(* Logix 5000 project; controller cal1632 1756-L62 rev 16.20; software revision 16.05; part 47 of 57 *)
(* tags used below, declared in another part *)
   FAULT : BOOL;
   HMI : BOOL;
   p01r09_pb_global_reset : BOOL;
   p02_dint_from_hmi : hmi_dint;
   p27_ao_dia_a : REAL;
   p27_ao_dia_b : REAL;
   p27_dint_to_hmi : DINT[16];
   p27_real_to_hmi : REAL[112];
   p27r05_lla_mode_tension : BOOL;
   p27r05_llb_mode_tension : BOOL;
   p27r06 : routine;
   p27r06_timer_fault : TIMER[4];
   p27r06_timer_warning : TIMER[4];
   p27r07 : routine;
   p27r07_timer_fault : TIMER[4];
   p27r07_timer_warning : TIMER[4];
   p27r08 : routine;
   p27r08_timer_fault : TIMER[4];
   p27r08_timer_warning : TIMER[4];
   p27r09 : routine;
   p27r09_a_enable_toggle : SYS_Toggle;
   p27r09_b_enable_toggle : SYS_Toggle;
   p27r09_timer_fault : TIMER[4];
   p27r09_timer_warning : TIMER[4];
(* P27_Lower_Poly_Letoff, continued *)

ROUTINE R06_Real_to_HMI   (* ladder *)
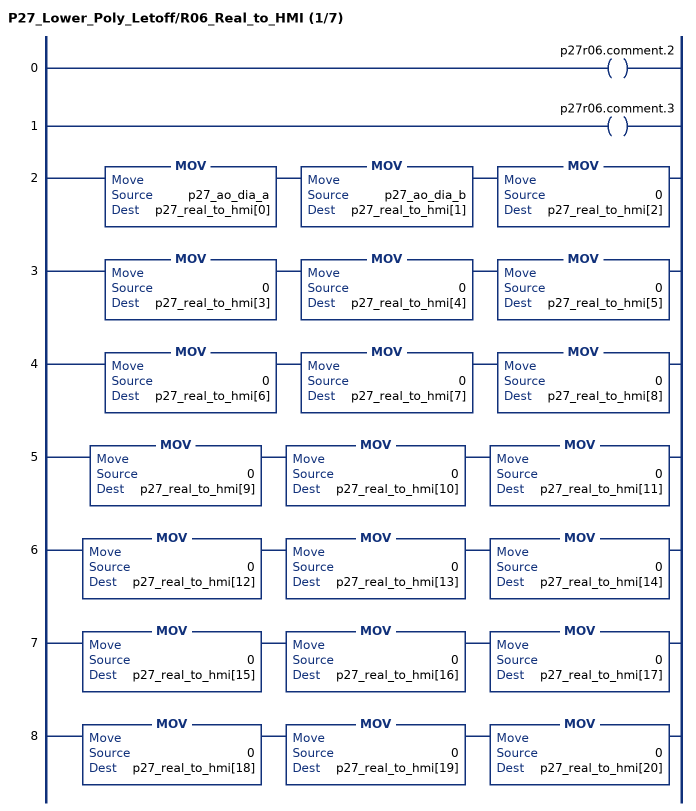
   0: OTE(p27r06.comment.2);
   1: OTE(p27r06.comment.3);
   2: MOV(p27_ao_dia_a,p27_real_to_hmi[0])MOV(p27_ao_dia_b,p27_real_to_hmi[1])MOV(0,p27_real_to_hmi[2]);
   3: MOV(0,p27_real_to_hmi[3])MOV(0,p27_real_to_hmi[4])MOV(0,p27_real_to_hmi[5]);
   4: MOV(0,p27_real_to_hmi[6])MOV(0,p27_real_to_hmi[7])MOV(0,p27_real_to_hmi[8]);
   5: MOV(0,p27_real_to_hmi[9])MOV(0,p27_real_to_hmi[10])MOV(0,p27_real_to_hmi[11]);
   6: MOV(0,p27_real_to_hmi[12])MOV(0,p27_real_to_hmi[13])MOV(0,p27_real_to_hmi[14]);
   7: MOV(0,p27_real_to_hmi[15])MOV(0,p27_real_to_hmi[16])MOV(0,p27_real_to_hmi[17]);
   8: MOV(0,p27_real_to_hmi[18])MOV(0,p27_real_to_hmi[19])MOV(0,p27_real_to_hmi[20]);
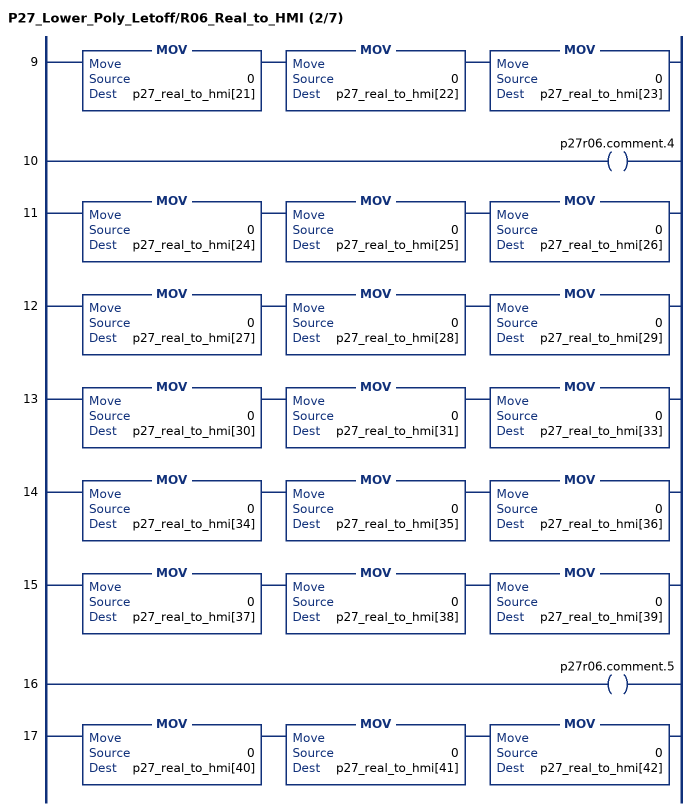
   9: MOV(0,p27_real_to_hmi[21])MOV(0,p27_real_to_hmi[22])MOV(0,p27_real_to_hmi[23]);
   10: OTE(p27r06.comment.4);
   11: MOV(0,p27_real_to_hmi[24])MOV(0,p27_real_to_hmi[25])MOV(0,p27_real_to_hmi[26]);
   12: MOV(0,p27_real_to_hmi[27])MOV(0,p27_real_to_hmi[28])MOV(0,p27_real_to_hmi[29]);
   13: MOV(0,p27_real_to_hmi[30])MOV(0,p27_real_to_hmi[31])MOV(0,p27_real_to_hmi[33]);
   14: MOV(0,p27_real_to_hmi[34])MOV(0,p27_real_to_hmi[35])MOV(0,p27_real_to_hmi[36]);
   15: MOV(0,p27_real_to_hmi[37])MOV(0,p27_real_to_hmi[38])MOV(0,p27_real_to_hmi[39]);
   16: OTE(p27r06.comment.5);
   17: MOV(0,p27_real_to_hmi[40])MOV(0,p27_real_to_hmi[41])MOV(0,p27_real_to_hmi[42]);
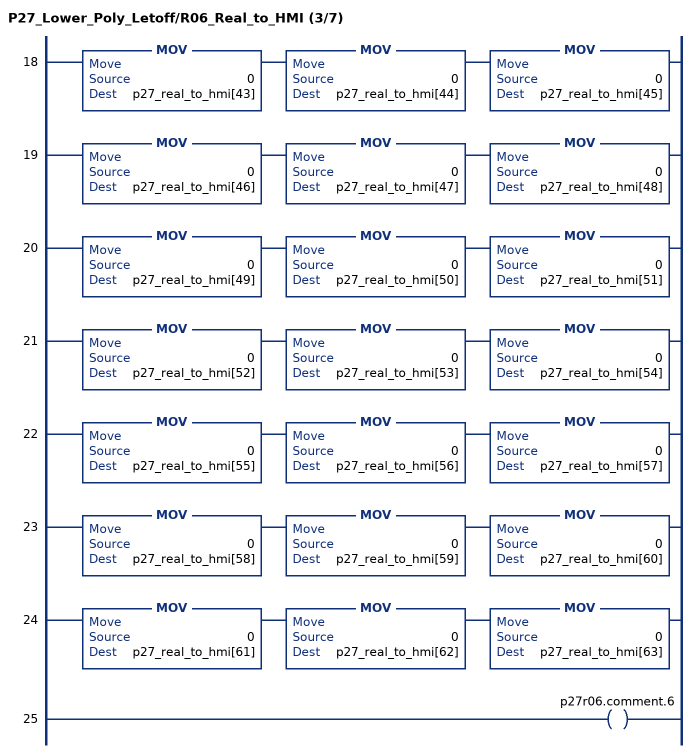
   18: MOV(0,p27_real_to_hmi[43])MOV(0,p27_real_to_hmi[44])MOV(0,p27_real_to_hmi[45]);
   19: MOV(0,p27_real_to_hmi[46])MOV(0,p27_real_to_hmi[47])MOV(0,p27_real_to_hmi[48]);
   20: MOV(0,p27_real_to_hmi[49])MOV(0,p27_real_to_hmi[50])MOV(0,p27_real_to_hmi[51]);
   21: MOV(0,p27_real_to_hmi[52])MOV(0,p27_real_to_hmi[53])MOV(0,p27_real_to_hmi[54]);
   22: MOV(0,p27_real_to_hmi[55])MOV(0,p27_real_to_hmi[56])MOV(0,p27_real_to_hmi[57]);
   23: MOV(0,p27_real_to_hmi[58])MOV(0,p27_real_to_hmi[59])MOV(0,p27_real_to_hmi[60]);
   24: MOV(0,p27_real_to_hmi[61])MOV(0,p27_real_to_hmi[62])MOV(0,p27_real_to_hmi[63]);
   25: OTE(p27r06.comment.6);
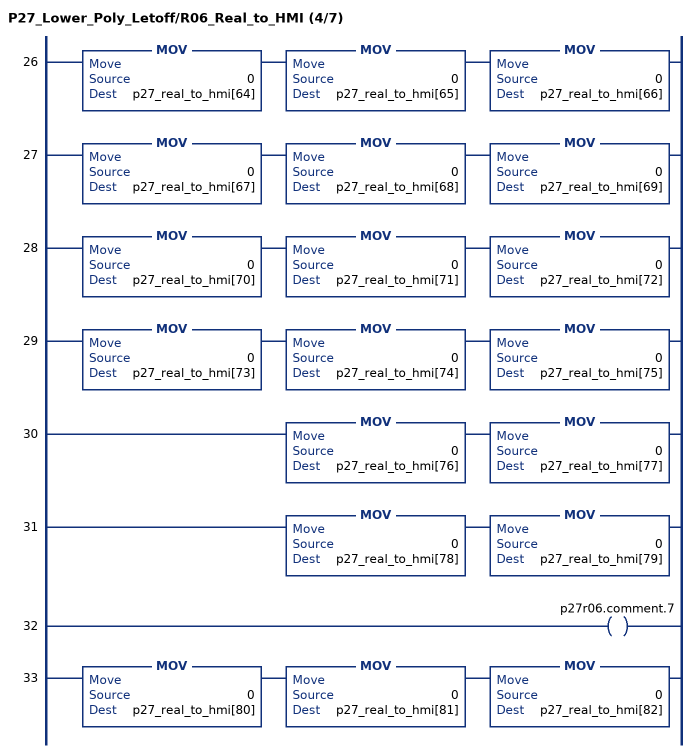
   26: MOV(0,p27_real_to_hmi[64])MOV(0,p27_real_to_hmi[65])MOV(0,p27_real_to_hmi[66]);
   27: MOV(0,p27_real_to_hmi[67])MOV(0,p27_real_to_hmi[68])MOV(0,p27_real_to_hmi[69]);
   28: MOV(0,p27_real_to_hmi[70])MOV(0,p27_real_to_hmi[71])MOV(0,p27_real_to_hmi[72]);
   29: MOV(0,p27_real_to_hmi[73])MOV(0,p27_real_to_hmi[74])MOV(0,p27_real_to_hmi[75]);
   30: MOV(0,p27_real_to_hmi[76])MOV(0,p27_real_to_hmi[77]);
   31: MOV(0,p27_real_to_hmi[78])MOV(0,p27_real_to_hmi[79]);
   32: OTE(p27r06.comment.7);
   33: MOV(0,p27_real_to_hmi[80])MOV(0,p27_real_to_hmi[81])MOV(0,p27_real_to_hmi[82]);
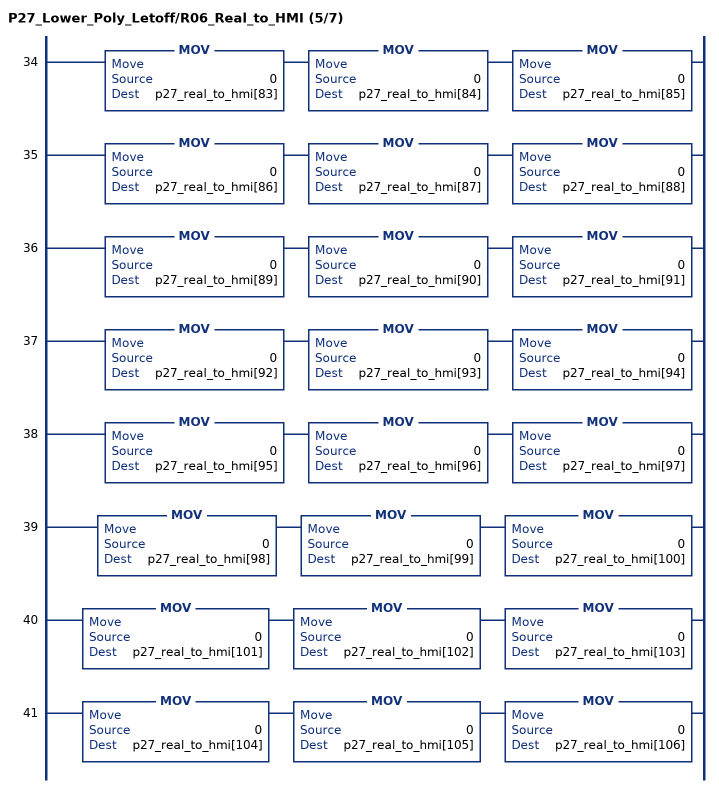
   34: MOV(0,p27_real_to_hmi[83])MOV(0,p27_real_to_hmi[84])MOV(0,p27_real_to_hmi[85]);
   35: MOV(0,p27_real_to_hmi[86])MOV(0,p27_real_to_hmi[87])MOV(0,p27_real_to_hmi[88]);
   36: MOV(0,p27_real_to_hmi[89])MOV(0,p27_real_to_hmi[90])MOV(0,p27_real_to_hmi[91]);
   37: MOV(0,p27_real_to_hmi[92])MOV(0,p27_real_to_hmi[93])MOV(0,p27_real_to_hmi[94]);
   38: MOV(0,p27_real_to_hmi[95])MOV(0,p27_real_to_hmi[96])MOV(0,p27_real_to_hmi[97]);
   39: MOV(0,p27_real_to_hmi[98])MOV(0,p27_real_to_hmi[99])MOV(0,p27_real_to_hmi[100]);
   40: MOV(0,p27_real_to_hmi[101])MOV(0,p27_real_to_hmi[102])MOV(0,p27_real_to_hmi[103]);
   41: MOV(0,p27_real_to_hmi[104])MOV(0,p27_real_to_hmi[105])MOV(0,p27_real_to_hmi[106]);
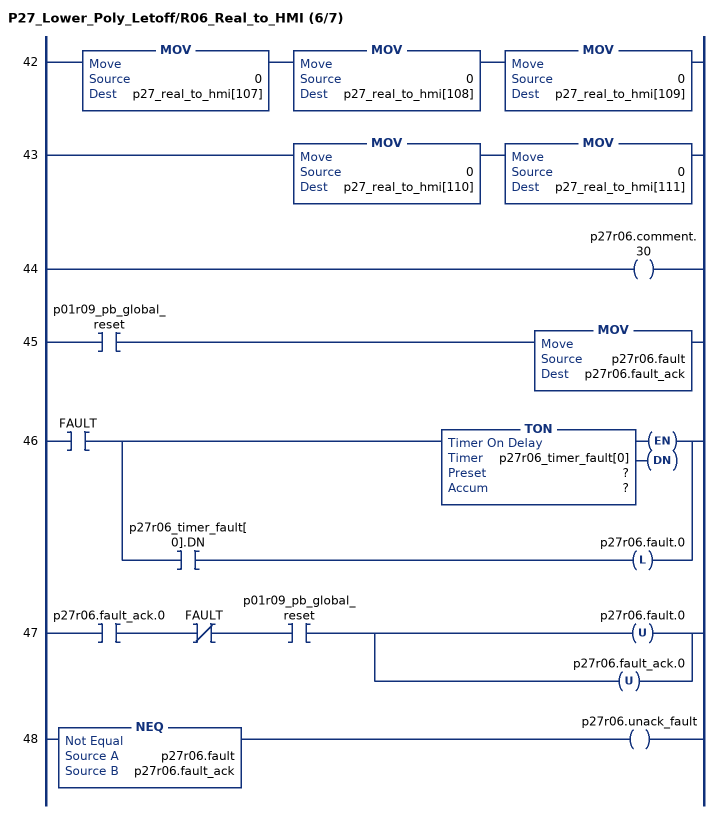
   42: MOV(0,p27_real_to_hmi[107])MOV(0,p27_real_to_hmi[108])MOV(0,p27_real_to_hmi[109]);
   43: MOV(0,p27_real_to_hmi[110])MOV(0,p27_real_to_hmi[111]);
   44: OTE(p27r06.comment.30);
   45: XIC(p01r09_pb_global_reset)MOV(p27r06.fault,p27r06.fault_ack);
   46: XIC(FAULT)[TON(p27r06_timer_fault[0],?,?) ,XIC(p27r06_timer_fault[0].DN) OTL(p27r06.fault.0) ];
   47: XIC(p27r06.fault_ack.0)XIO(FAULT)XIC(p01r09_pb_global_reset)[OTU(p27r06.fault.0) ,OTU(p27r06.fault_ack.0) ];
   48: NEQ(p27r06.fault,p27r06.fault_ack)OTE(p27r06.unack_fault);
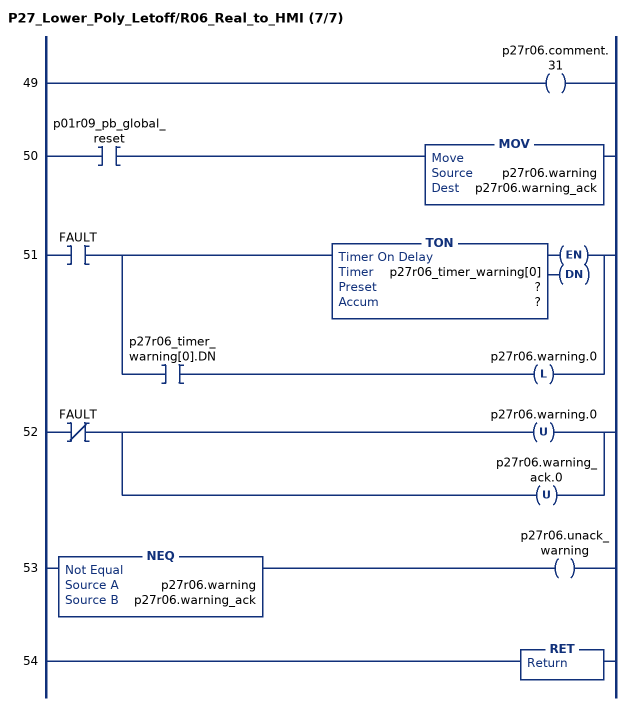
   49: OTE(p27r06.comment.31);
   50: XIC(p01r09_pb_global_reset)MOV(p27r06.warning,p27r06.warning_ack);
   51: XIC(FAULT)[TON(p27r06_timer_warning[0],?,?) ,XIC(p27r06_timer_warning[0].DN) OTL(p27r06.warning.0) ];
   52: XIO(FAULT)[OTU(p27r06.warning.0) ,OTU(p27r06.warning_ack.0) ];
   53: NEQ(p27r06.warning,p27r06.warning_ack)OTE(p27r06.unack_warning);
   54: RET();
END_ROUTINE

ROUTINE R07_Alarms   (* ladder *)
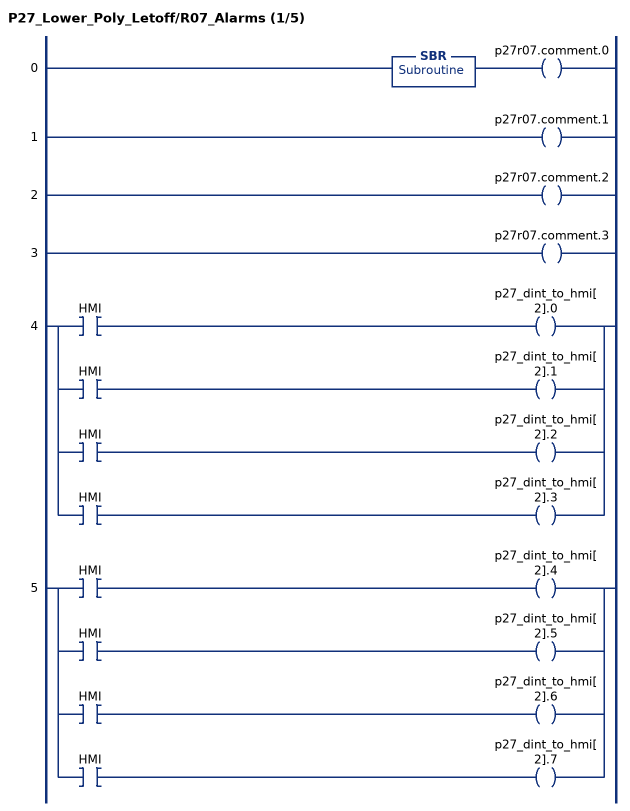
   0: SBR()OTE(p27r07.comment.0);
   1: OTE(p27r07.comment.1);
   2: OTE(p27r07.comment.2);
   3: OTE(p27r07.comment.3);
   4: [XIC(HMI) OTE(p27_dint_to_hmi[2].0) ,XIC(HMI) OTE(p27_dint_to_hmi[2].1) ,XIC(HMI) OTE(p27_dint_to_hmi[2].2) ,XIC(HMI) OTE(p27_dint_to_hmi[2].3) ];
   5: [XIC(HMI) OTE(p27_dint_to_hmi[2].4) ,XIC(HMI) OTE(p27_dint_to_hmi[2].5) ,XIC(HMI) OTE(p27_dint_to_hmi[2].6) ,XIC(HMI) OTE(p27_dint_to_hmi[2].7) ];
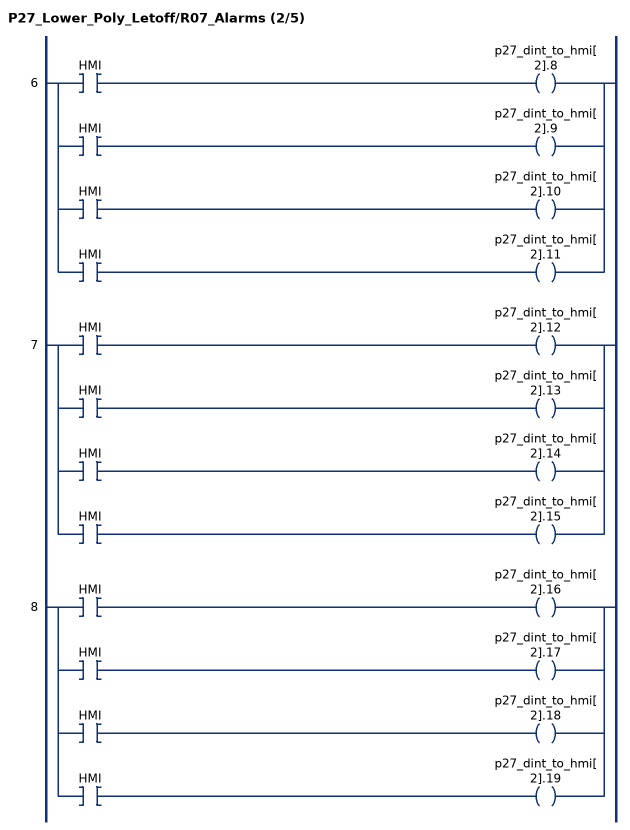
   6: [XIC(HMI) OTE(p27_dint_to_hmi[2].8) ,XIC(HMI) OTE(p27_dint_to_hmi[2].9) ,XIC(HMI) OTE(p27_dint_to_hmi[2].10) ,XIC(HMI) OTE(p27_dint_to_hmi[2].11) ];
   7: [XIC(HMI) OTE(p27_dint_to_hmi[2].12) ,XIC(HMI) OTE(p27_dint_to_hmi[2].13) ,XIC(HMI) OTE(p27_dint_to_hmi[2].14) ,XIC(HMI) OTE(p27_dint_to_hmi[2].15) ];
   8: [XIC(HMI) OTE(p27_dint_to_hmi[2].16) ,XIC(HMI) OTE(p27_dint_to_hmi[2].17) ,XIC(HMI) OTE(p27_dint_to_hmi[2].18) ,XIC(HMI) OTE(p27_dint_to_hmi[2].19) ];
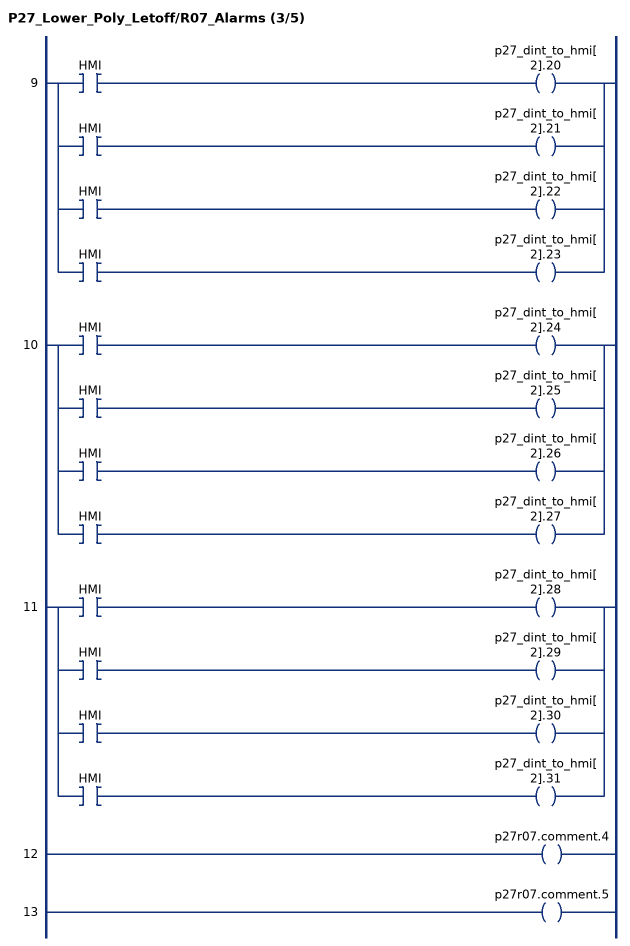
   9: [XIC(HMI) OTE(p27_dint_to_hmi[2].20) ,XIC(HMI) OTE(p27_dint_to_hmi[2].21) ,XIC(HMI) OTE(p27_dint_to_hmi[2].22) ,XIC(HMI) OTE(p27_dint_to_hmi[2].23) ];
   10: [XIC(HMI) OTE(p27_dint_to_hmi[2].24) ,XIC(HMI) OTE(p27_dint_to_hmi[2].25) ,XIC(HMI) OTE(p27_dint_to_hmi[2].26) ,XIC(HMI) OTE(p27_dint_to_hmi[2].27) ];
   11: [XIC(HMI) OTE(p27_dint_to_hmi[2].28) ,XIC(HMI) OTE(p27_dint_to_hmi[2].29) ,XIC(HMI) OTE(p27_dint_to_hmi[2].30) ,XIC(HMI) OTE(p27_dint_to_hmi[2].31) ];
   12: OTE(p27r07.comment.4);
   13: OTE(p27r07.comment.5);
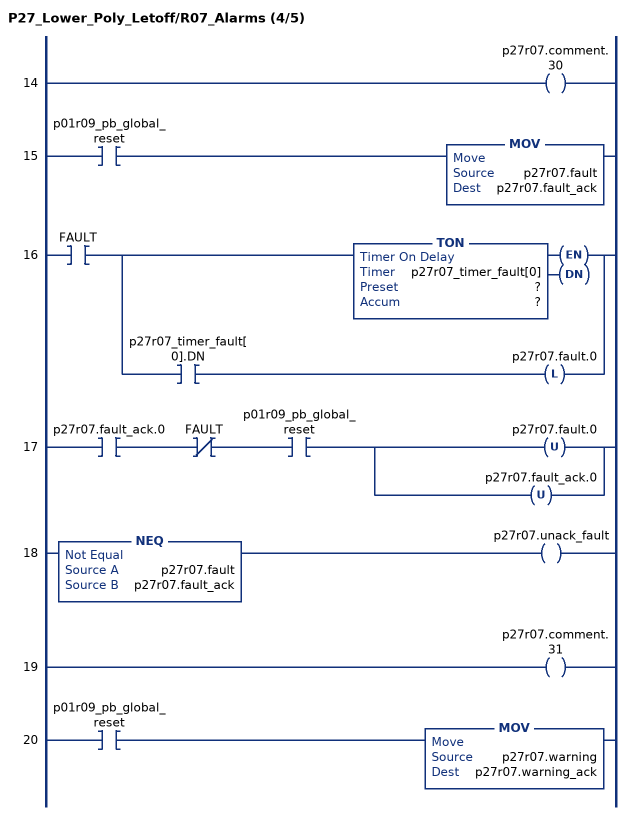
   14: OTE(p27r07.comment.30);
   15: XIC(p01r09_pb_global_reset)MOV(p27r07.fault,p27r07.fault_ack);
   16: XIC(FAULT)[TON(p27r07_timer_fault[0],?,?) ,XIC(p27r07_timer_fault[0].DN) OTL(p27r07.fault.0) ];
   17: XIC(p27r07.fault_ack.0)XIO(FAULT)XIC(p01r09_pb_global_reset)[OTU(p27r07.fault.0) ,OTU(p27r07.fault_ack.0) ];
   18: NEQ(p27r07.fault,p27r07.fault_ack)OTE(p27r07.unack_fault);
   19: OTE(p27r07.comment.31);
   20: XIC(p01r09_pb_global_reset)MOV(p27r07.warning,p27r07.warning_ack);
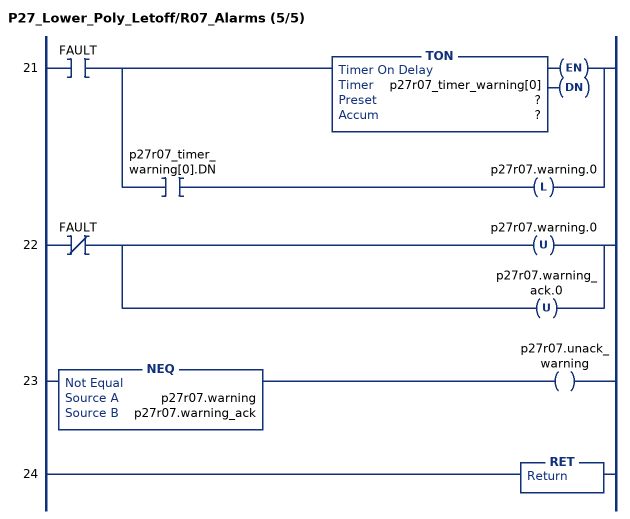
   21: XIC(FAULT)[TON(p27r07_timer_warning[0],?,?) ,XIC(p27r07_timer_warning[0].DN) OTL(p27r07.warning.0) ];
   22: XIO(FAULT)[OTU(p27r07.warning.0) ,OTU(p27r07.warning_ack.0) ];
   23: NEQ(p27r07.warning,p27r07.warning_ack)OTE(p27r07.unack_warning);
   24: RET();
END_ROUTINE

ROUTINE R08_Warnings   (* ladder *)
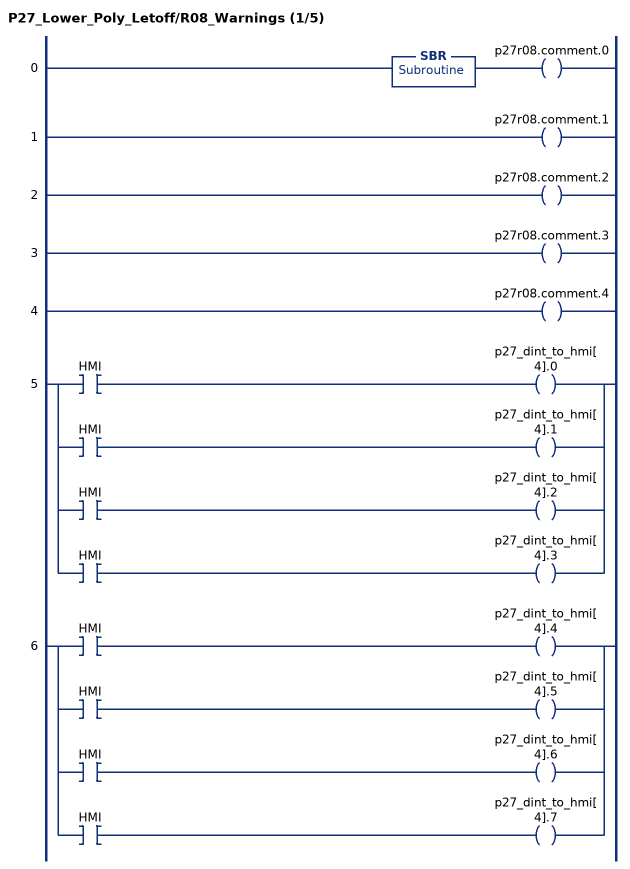
   0: SBR()OTE(p27r08.comment.0);
   1: OTE(p27r08.comment.1);
   2: OTE(p27r08.comment.2);
   3: OTE(p27r08.comment.3);
   4: OTE(p27r08.comment.4);
   5: [XIC(HMI) OTE(p27_dint_to_hmi[4].0) ,XIC(HMI) OTE(p27_dint_to_hmi[4].1) ,XIC(HMI) OTE(p27_dint_to_hmi[4].2) ,XIC(HMI) OTE(p27_dint_to_hmi[4].3) ];
   6: [XIC(HMI) OTE(p27_dint_to_hmi[4].4) ,XIC(HMI) OTE(p27_dint_to_hmi[4].5) ,XIC(HMI) OTE(p27_dint_to_hmi[4].6) ,XIC(HMI) OTE(p27_dint_to_hmi[4].7) ];
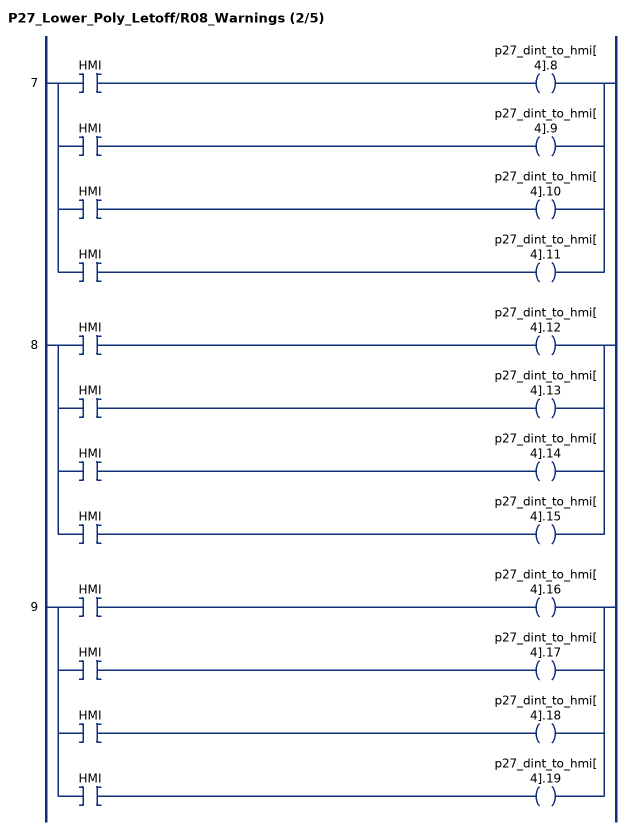
   7: [XIC(HMI) OTE(p27_dint_to_hmi[4].8) ,XIC(HMI) OTE(p27_dint_to_hmi[4].9) ,XIC(HMI) OTE(p27_dint_to_hmi[4].10) ,XIC(HMI) OTE(p27_dint_to_hmi[4].11) ];
   8: [XIC(HMI) OTE(p27_dint_to_hmi[4].12) ,XIC(HMI) OTE(p27_dint_to_hmi[4].13) ,XIC(HMI) OTE(p27_dint_to_hmi[4].14) ,XIC(HMI) OTE(p27_dint_to_hmi[4].15) ];
   9: [XIC(HMI) OTE(p27_dint_to_hmi[4].16) ,XIC(HMI) OTE(p27_dint_to_hmi[4].17) ,XIC(HMI) OTE(p27_dint_to_hmi[4].18) ,XIC(HMI) OTE(p27_dint_to_hmi[4].19) ];
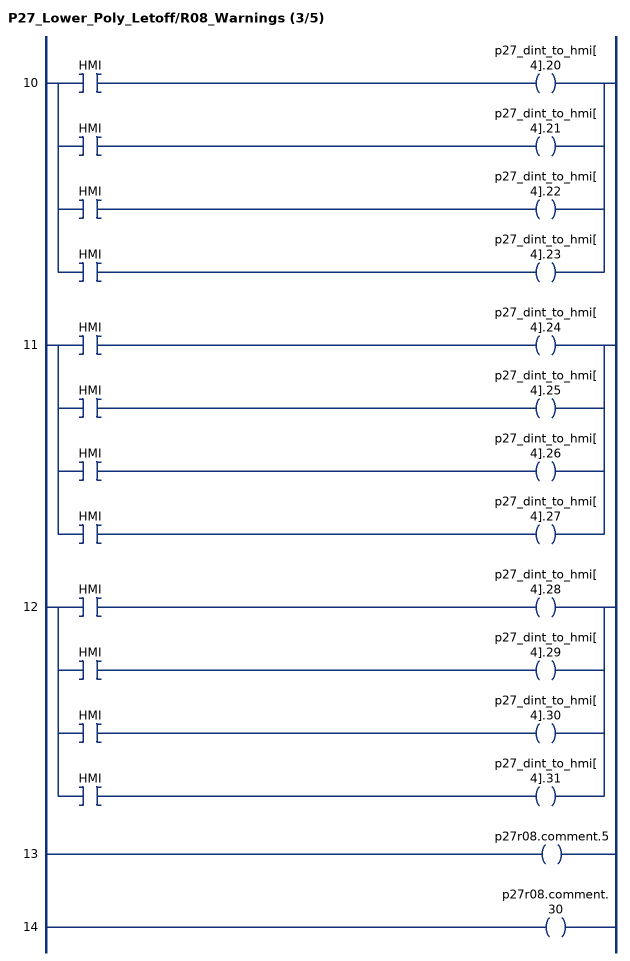
   10: [XIC(HMI) OTE(p27_dint_to_hmi[4].20) ,XIC(HMI) OTE(p27_dint_to_hmi[4].21) ,XIC(HMI) OTE(p27_dint_to_hmi[4].22) ,XIC(HMI) OTE(p27_dint_to_hmi[4].23) ];
   11: [XIC(HMI) OTE(p27_dint_to_hmi[4].24) ,XIC(HMI) OTE(p27_dint_to_hmi[4].25) ,XIC(HMI) OTE(p27_dint_to_hmi[4].26) ,XIC(HMI) OTE(p27_dint_to_hmi[4].27) ];
   12: [XIC(HMI) OTE(p27_dint_to_hmi[4].28) ,XIC(HMI) OTE(p27_dint_to_hmi[4].29) ,XIC(HMI) OTE(p27_dint_to_hmi[4].30) ,XIC(HMI) OTE(p27_dint_to_hmi[4].31) ];
   13: OTE(p27r08.comment.5);
   14: OTE(p27r08.comment.30);
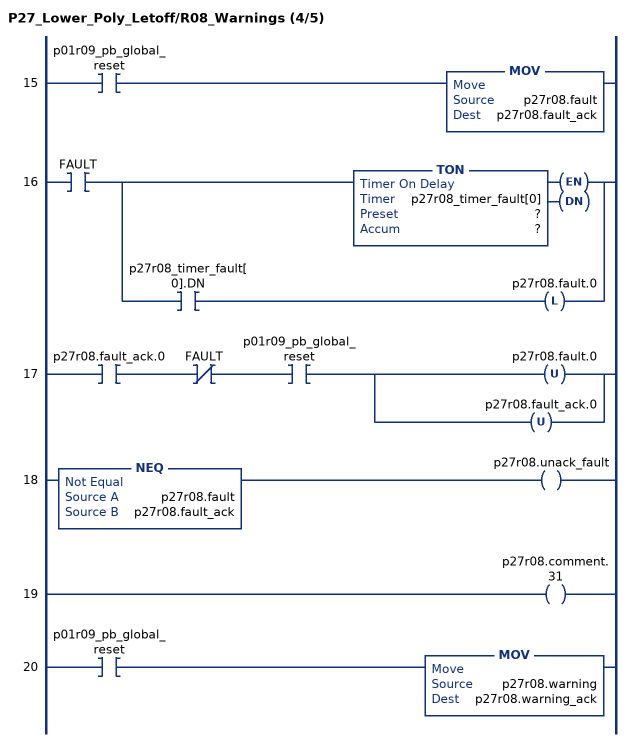
   15: XIC(p01r09_pb_global_reset)MOV(p27r08.fault,p27r08.fault_ack);
   16: XIC(FAULT)[TON(p27r08_timer_fault[0],?,?) ,XIC(p27r08_timer_fault[0].DN) OTL(p27r08.fault.0) ];
   17: XIC(p27r08.fault_ack.0)XIO(FAULT)XIC(p01r09_pb_global_reset)[OTU(p27r08.fault.0) ,OTU(p27r08.fault_ack.0) ];
   18: NEQ(p27r08.fault,p27r08.fault_ack)OTE(p27r08.unack_fault);
   19: OTE(p27r08.comment.31);
   20: XIC(p01r09_pb_global_reset)MOV(p27r08.warning,p27r08.warning_ack);
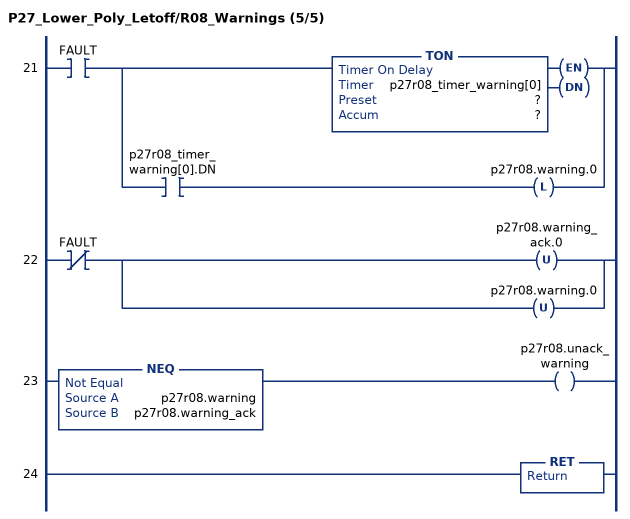
   21: XIC(FAULT)[TON(p27r08_timer_warning[0],?,?) ,XIC(p27r08_timer_warning[0].DN) OTL(p27r08.warning.0) ];
   22: XIO(FAULT)[OTU(p27r08.warning_ack.0) ,OTU(p27r08.warning.0) ];
   23: NEQ(p27r08.warning,p27r08.warning_ack)OTE(p27r08.unack_warning);
   24: RET();
END_ROUTINE

ROUTINE R09_Modes   (* ladder *)
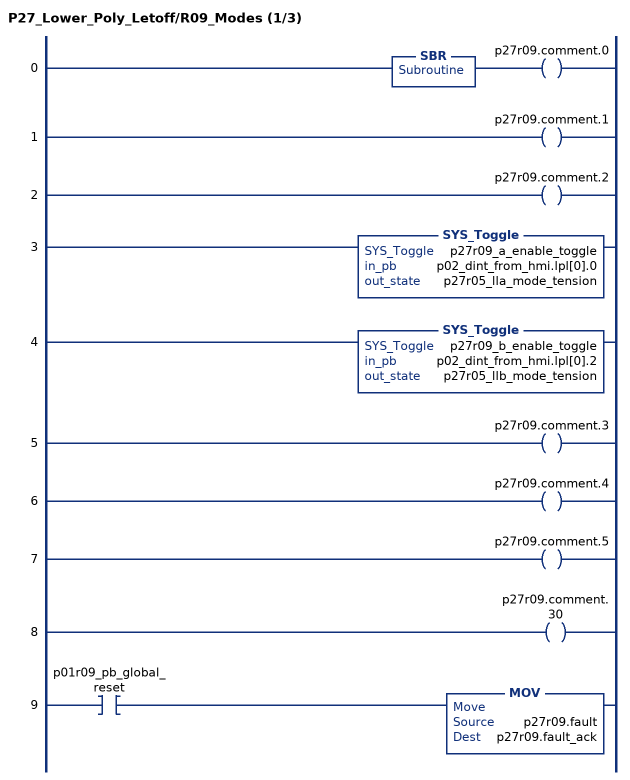
   0: SBR()OTE(p27r09.comment.0);
   1: OTE(p27r09.comment.1);
   2: OTE(p27r09.comment.2);
   3: SYS_Toggle(p27r09_a_enable_toggle,p02_dint_from_hmi.lpl[0].0,p27r05_lla_mode_tension);
   4: SYS_Toggle(p27r09_b_enable_toggle,p02_dint_from_hmi.lpl[0].2,p27r05_llb_mode_tension);
   5: OTE(p27r09.comment.3);
   6: OTE(p27r09.comment.4);
   7: OTE(p27r09.comment.5);
   8: OTE(p27r09.comment.30);
   9: XIC(p01r09_pb_global_reset)MOV(p27r09.fault,p27r09.fault_ack);
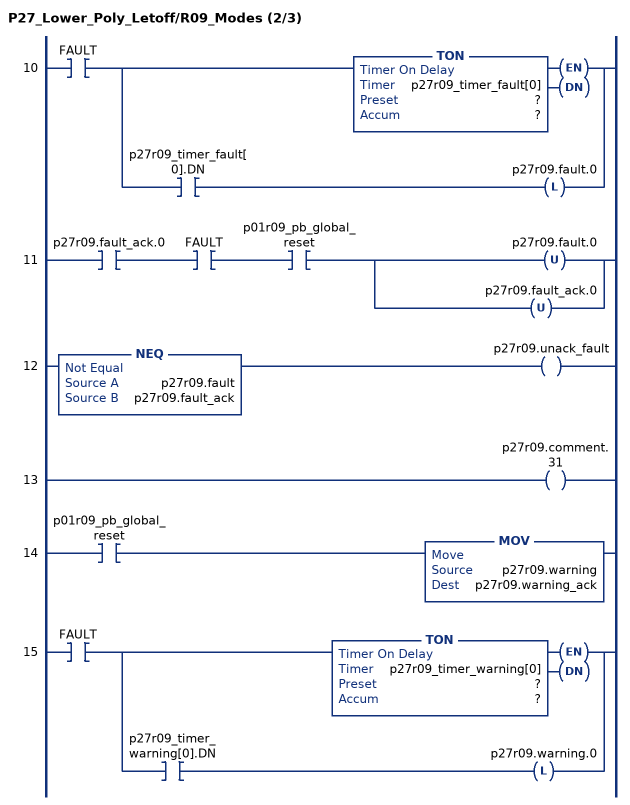
   10: XIC(FAULT)[TON(p27r09_timer_fault[0],?,?) ,XIC(p27r09_timer_fault[0].DN) OTL(p27r09.fault.0) ];
   11: XIC(p27r09.fault_ack.0)XIC(FAULT)XIC(p01r09_pb_global_reset)[OTU(p27r09.fault.0) ,OTU(p27r09.fault_ack.0) ];
   12: NEQ(p27r09.fault,p27r09.fault_ack)OTE(p27r09.unack_fault);
   13: OTE(p27r09.comment.31);
   14: XIC(p01r09_pb_global_reset)MOV(p27r09.warning,p27r09.warning_ack);
   15: XIC(FAULT)[TON(p27r09_timer_warning[0],?,?) ,XIC(p27r09_timer_warning[0].DN) OTL(p27r09.warning.0) ];
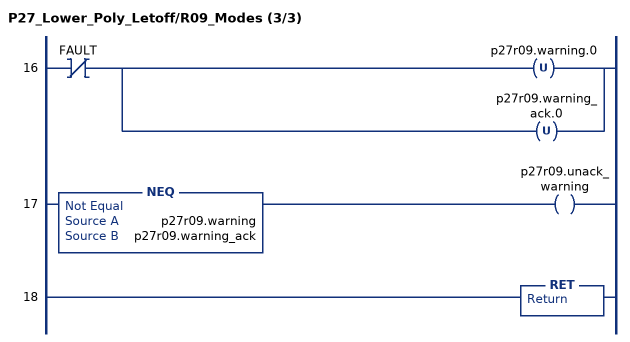
   16: XIO(FAULT)[OTU(p27r09.warning.0) ,OTU(p27r09.warning_ack.0) ];
   17: NEQ(p27r09.warning,p27r09.warning_ack)OTE(p27r09.unack_warning);
   18: RET();
END_ROUTINE
